PROGRAM Conveyor_Controller
  VAR_EXTERNAL
    Safety_OK : BOOL;
    Conveyor_Start : BOOL;
    Conveyor_Stop : BOOL;
    System_Reset : BOOL;
    Auto_Request : BOOL;
  END_VAR
  VAR
    Conveyor_Auto : BOOL;
    Conveyor_Start_Cmd : BOOL;
    Conveyor_Stop_Cmd : BOOL;
    Conveyor_Jam : BOOL;
    Conveyor_Run : BOOL;
    Conveyor_Jam_Timer : TON;
    Entry_Sensor : BOOL;
    Exit_Sensor : BOOL;
  END_VAR

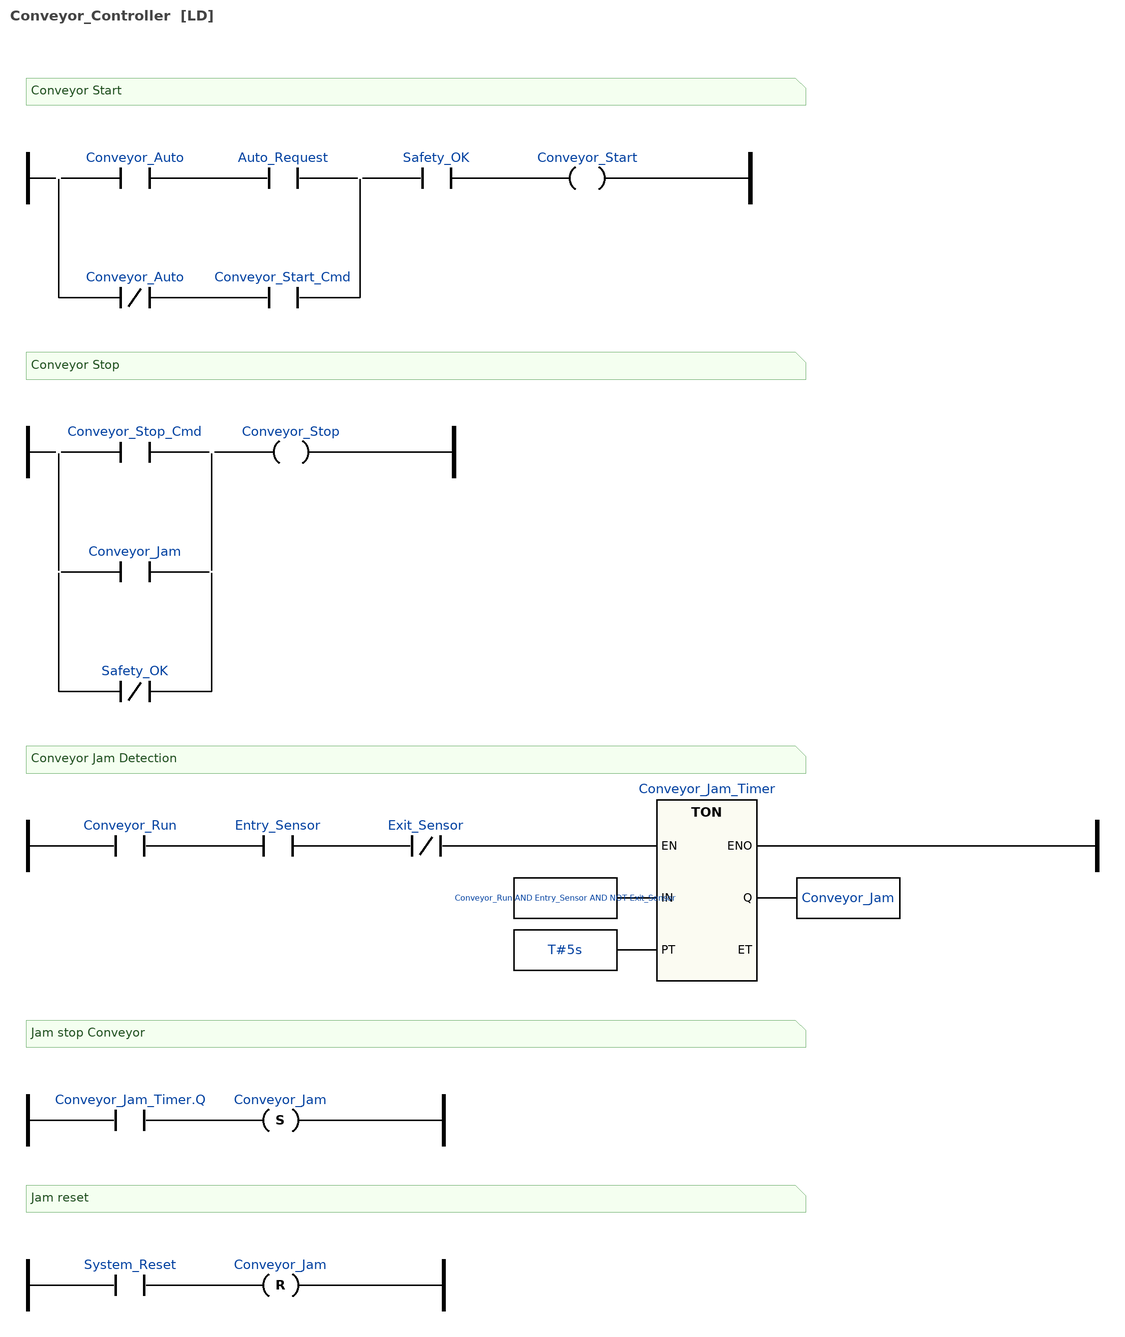
(* LD diagram, written out as Structured Text *)
(* Conveyor Start *)
Conveyor_Start := (NOT Conveyor_Auto AND Conveyor_Start_Cmd OR Conveyor_Auto AND Auto_Request) AND Safety_OK;
(* Conveyor Stop *)
Conveyor_Stop := Conveyor_Stop_Cmd OR Conveyor_Jam OR NOT Safety_OK;
(* Conveyor Jam Detection *)
Conveyor_Jam_Timer(EN := Conveyor_Run AND Entry_Sensor AND NOT Exit_Sensor, IN := Conveyor_Run AND Entry_Sensor AND NOT Exit_Sensor, PT := T#5s);
IF Conveyor_Jam_Timer.ENO THEN Conveyor_Jam := Conveyor_Jam_Timer.Q; END_IF;
(* Jam stop Conveyor *)
IF Conveyor_Jam_Timer.Q THEN Conveyor_Jam := TRUE; END_IF;
(* Jam reset *)
IF System_Reset THEN Conveyor_Jam := FALSE; END_IF;
END_PROGRAM
